KUKA KRL program: MIN.src

&ACCESS RV1
&REL 1
&PARAM TEMPLATE = C:\KRC\Roboter\Template\FunctionVorgabe
&PARAM EDITMASK = *
DEFFCT REAL MIN(VALUE1:IN, VALUE2:IN )
  REAL VALUE1
  REAL VALUE2
  REAL RET_VAL

  IF VALUE1 > VALUE2 THEN
    RET_VAL = VALUE2
  ELSE
    RET_VAL = VALUE1
  ENDIF

  RETURN(RET_VAL)
ENDFCT
